// TwinCAT 3 PLC project Bohrmodell_SK1
// ProgramVersion: 3.1.4024.12
// libraries:
//   Tc2_EtherCAT, * (Beckhoff Automation GmbH)
//   Tc2_Standard, * (Beckhoff Automation GmbH)
//   Tc2_System, * (Beckhoff Automation GmbH)
//   Tc3_Module, * (Beckhoff Automation GmbH)
//   VisuSymbols,3.5.10.0,System
// project tree:
//   DUTs/ DUT_Motordaten.TcDUT, E_AmpelPhase.TcDUT, E_BMK.TcDUT, E_Step.TcDUT, ST_Test.TcDUT
//   / GlobalTextList.TcGTLO, PlcTask.TcTTO, TaktGen.TcTTO, Visualisierungsmanager.TcVMO (not stored)
//   GVLs/ GVL_Datenverarbeitung.TcGVL, GVL_GK_Automatikablauf.TcGVL, GVL_GlobalData.TcGVL, GVL_A1.TcGVL, GVL_C1.TcGVL, GVL_HMI.TcGVL
//   POUs/Ampelsteuerung/ DUT_AmpelConfig.TcDUT, E_Ampeln.TcDUT, FB_Ampel.TcPOU, GVL_Ampel.TcGVL, GVL_HMI_Ampel.TcGVL
//   POUs/Funktionen/ FB_Counter.TcPOU
//   POUs/HMI/ PRG_HMI.TcPOU
//   POUs/Mod01_Allgm/ FB_BA_Umschaltung_FUP.TcPOU, PRG_TaktGen.TcPOU, FB_BA_Umschaltung.TcPOU
//   POUs/Mod03_Diag/ FB_AdsLog.TcPOU
//   POUs/Mod20_Analog/ FB_Tank.TcPOU
//   POUs/ FB_StrukturieterText.TcPOU, POU_ST_FUP.TcPOU, PRG_MAIN.TcPOU
//   POUs/Geraete/ FB_Betriebsarten.TcPOU, FB_Motor.TcPOU
//   POUs/Mod10_FT/ FB_Antriebe.TcPOU, FB_Autoamtikablauf.TcPOU
//   POUs/Mod30/ FB_Refactoring.TcPOU, FB_RefDummy.TcPOU
//   POUs/TOOLS/ FB_Takt.TcPOU
//   VISUs/ Ampel.TcVIS, FP_Counter.TcVIS, Visualization.TcVIS
//   VISUs/Pages/ Page_2.TcVIS, Page_3.TcVIS
//   VISUs/Tempalte/ Visualization_1.TcVIS
// real-time tasks:
//   TASK PlcTask: cycle T#10ms, priority 6, ADS port 350
//   TASK TaktGen: cycle T#10ms, priority 8, ADS port 351
// I/O:
//   DEVICE Gerät 2 (EtherCAT), AmsNetId 172.16.0.8.3.1
//     Klemme 1 (EK1200) [EK1200-5000 EtherCAT Netzteil (2A E-Bus)]
//       -KF2 (EL1809) [EL1809 16K. Dig. Eingang 24V, 3ms]
//       Klemme 3 (EL1809) [EL1809 16K. Dig. Eingang 24V, 3ms]
//       Klemme 4 (EL2809) [EL2809 16K. Dig. Ausgang 24V, 0.5A]
//       Klemme 5 (EL2809) [EL2809 16K. Dig. Ausgang 24V, 0.5A]
//       Klemme 6 (EK1110) [EK1110 EtherCAT-Verlängerung]
//     Klemme 7 (EK1100) [EK1100 EtherCAT-Koppler (2A E-Bus)]
//       Klemme 8 (EL3062) [EL3062 2K.Ana. Eingang 0-10V]
//       Klemme 9 (EL4002) [EL4002 2K. Ana. Ausgang 0-10V, 12bit]
//       Klemme 10 (EL9011) [EL9011 Endklemme]
//     Box 20 (TB20 Coupler EtherCAT) [TB20 Coupler EtherCAT (600-185-1AA11)]
//       modules: Module 1 (8 DI - 600-210-0AH01), Module 2 (8 DO - 600-220-0AH01)
// variable links:
//   Bohrmodell_SK1/Bohrmodell_SK1 Instance <-> Device 2 (EtherCAT)/Term 1 (EK1200)/-KF2 (EL1809)
//     PlcTask Inputs/GVL_A1.GL1_B1_BG1 <-> Channel 9/GL1_B1_BG1
//     PlcTask Inputs/GVL_A1.GL2_B2_BG1 <-> Channel 10/GL2_B2_BG1
//     PlcTask Inputs/GVL_A1.GL3_B3_BG1 <-> Channel 11/Input
//     PlcTask Inputs/GVL_A1.TM1_B2_BG1 <-> Channel 12/Input
//     PlcTask Inputs/GVL_A1.TM1_B2_BG2 <-> Channel 13/Input
//     TaktGen Inputs/GVL_A1.GL1_B1_BQ1 <-> Channel 16/Input
//     TaktGen Inputs/GVL_A1.S01_C2_SF1 <-> Channel 14/Input
//     TaktGen Inputs/GVL_A1.S01_C3_SF1 <-> Channel 15/Input
//   Bohrmodell_SK1/Bohrmodell_SK1 Instance <-> Device 2 (EtherCAT)/Term 1 (EK1200)/Term 3 (EL1809)
//     PlcTask Inputs/GVL_C1.S01_C1_SF1 <-> Channel 1/S01_C1_SF1
//     PlcTask Inputs/GVL_C1.S01_C1_SF2 <-> Channel 2/S01_C1_SF2
//     PlcTask Inputs/GVL_C1.S01_C1_SF10 <-> Channel 10/Input
//     PlcTask Inputs/GVL_C1.S01_C1_SF11 <-> Channel 11/Input
//     PlcTask Inputs/GVL_C1.S01_C1_SF12 <-> Channel 12/Input
//     PlcTask Inputs/GVL_C1.S01_C1_SF13 <-> Channel 13/Input
//     PlcTask Inputs/GVL_C1.S01_C1_SF14 <-> Channel 14/Input
//     PlcTask Inputs/GVL_C1.S01_C1_SF16 <-> Channel 16/Input
//     PlcTask Inputs/GVL_C1.S01_C1_SF9 <-> Channel 9/Input
//     PlcTask Inputs/GVL_C1.S01_C1_SF3 <-> Channel 3/GVL_C1.S01_C1_SF3
//     TaktGen Inputs/GVL_C1.S01_C1_SF15 <-> Channel 15/Input
//     TaktGen Inputs/GVL_C1.S01_C1_SF6 <-> Channel 6/Input
//     TaktGen Inputs/GVL_C1.S01_C1_SF7 <-> Channel 7/Input
//     TaktGen Inputs/GVL_C1.S01_C1_SF8 <-> Channel 8/Input
//     TaktGen Inputs/GVL_C1.S01_C1_SF4 <-> Channel 4/GVL_C1.S01_C1_SF4
//     TaktGen Inputs/GVL_C1.S01_C1_SF5 <-> Channel 5/GVL_C1.S01_C1_SF5
//   Bohrmodell_SK1/Bohrmodell_SK1 Instance <-> Device 2 (EtherCAT)/Term 1 (EK1200)/Term 4 (EL2809)
//     PlcTask Outputs/GVL_A1.GL1_B1_MA1 <-> Channel 1/Output
//     PlcTask Outputs/GVL_A1.GL2_B2_MA1 <-> Channel 2/Output
//     PlcTask Outputs/GVL_A1.GL3_B3_MA1 <-> Channel 3/Output
//     PlcTask Outputs/GVL_A1.S01_C3_PF1 <-> Channel 11/Output
//     PlcTask Outputs/GVL_A1.S01_C3_PF2 <-> Channel 12/Output
//     PlcTask Outputs/GVL_A1.S01_C3_PF3 <-> Channel 13/Output
//     PlcTask Outputs/GVL_A1.S01_C3_PJ1 <-> Channel 15/Output
//     PlcTask Outputs/GVL_A1.TM1_B2_MA1 <-> Channel 4/Output
//     PlcTask Outputs/GVL_A1.TM1_B2_MA2_1 <-> Channel 5/Output
//     PlcTask Outputs/GVL_A1.TM1_B2_MA2_2 <-> Channel 6/Output
//     TaktGen Outputs/GVL_A1.S01_C2_PF1 <-> Channel 9/Output
//     TaktGen Outputs/GVL_A1.S01_C2_PF2 <-> Channel 10/Output
//     TaktGen Outputs/GVL_A1.S01_C3_PF4 <-> Channel 14/Output
//   Bohrmodell_SK1/Bohrmodell_SK1 Instance <-> Device 2 (EtherCAT)/Term 1 (EK1200)/Term 5 (EL2809)
//     PlcTask Outputs/GVL_C1.S01_C1_PF1 <-> Channel 1/Output
//     PlcTask Outputs/GVL_C1.S01_C1_PF10 <-> Channel 10/Output
//     PlcTask Outputs/GVL_C1.S01_C1_PF11 <-> Channel 11/Output
//     PlcTask Outputs/GVL_C1.S01_C1_PF15 <-> Channel 15/Output
//     PlcTask Outputs/GVL_C1.S01_C1_PF16 <-> Channel 16/Output
//     PlcTask Outputs/GVL_C1.S01_C1_PF2 <-> Channel 2/Output
//     PlcTask Outputs/GVL_C1.S01_C1_PF3 <-> Channel 3/Output
//     PlcTask Outputs/GVL_C1.S01_C1_PF4 <-> Channel 4/Output
//     PlcTask Outputs/GVL_C1.S01_C1_PF5 <-> Channel 5/Output
//     PlcTask Outputs/GVL_C1.S01_C1_PF6 <-> Channel 6/Output
//     PlcTask Outputs/GVL_C1.S01_C1_PF9 <-> Channel 9/Output
//     TaktGen Outputs/GVL_C1.S01_C1_PF12 <-> Channel 12/Output
//     TaktGen Outputs/GVL_C1.S01_C1_PF13 <-> Channel 13/Output
//     TaktGen Outputs/GVL_C1.S01_C1_PF14 <-> Channel 14/Output
//     TaktGen Outputs/GVL_C1.S01_C1_PF7 <-> Channel 7/Output
//     TaktGen Outputs/GVL_C1.S01_C1_PF8 <-> Channel 8/Output

CONFIGURATION Bohrmodell_SK1
    RESOURCE PLC ON TwinCAT3
        TASK PlcTask(INTERVAL := T#10ms, PRIORITY := 6);
        TASK TaktGen(INTERVAL := T#10ms, PRIORITY := 8);
        PROGRAM PRG_MAIN WITH PlcTask : PRG_MAIN;
        PROGRAM PRG_HMI WITH PlcTask : PRG_HMI;
        PROGRAM PRG_TaktGen WITH TaktGen : PRG_TaktGen;
    END_RESOURCE
END_CONFIGURATION

// ---- DUTs/DUT_Motordaten.TcDUT
TYPE DUT_Motordaten :
STRUCT
	Laufzeit : INT;
	Einschaltvorgange : UINT;
	Motorleistung : REAL;
	Motorstrom : REAL;
	Drehzahl : INT;
	ResetDisable : BOOL;
END_STRUCT
END_TYPE

// ---- DUTs/E_AmpelPhase.TcDUT
{attribute 'qualified_only'}
{attribute 'strict'}
TYPE E_AmpelPhase :
(
	INIT := 0,
	ROT,
	GRUEN,
	GELB,
	ROTGELB
);
END_TYPE

// ---- DUTs/E_BMK.TcDUT
{attribute 'qualified_only'}
{attribute 'strict'}
TYPE E_BMK :
(
	Band_1 := 1,
	Band_2 := 2,
	Band_3 := 3,
	Bohrer  := 4,	
	BW_FWD  := 5,
	BW_BWD  := 6
	
);
END_TYPE

// ---- DUTs/E_Step.TcDUT
{attribute 'qualified_only'}
{attribute 'strict'}
TYPE E_Step :
(
	START,
	STOP,
	DRILL_FWD,
	DRILL_BWD,
	FEED_IN,
	FEED_OUT,
	WAIT,
	IN_END_POS
	
);
END_TYPE

// ---- DUTs/ST_Test.TcDUT
TYPE ST_Test :
STRUCT
	var1: BOOL;
	var2: INT;
	VarArray: ARRAY [0..11] OF INT;
END_STRUCT
END_TYPE

// ---- POUs/Ampelsteuerung/DUT_AmpelConfig.TcDUT
TYPE DUT_AmpelConfig :
STRUCT
	tRot		:TIME; // Zet für die Rotphase
	tRotGelb	:TIME;	// Zeit für die RotGruenphase
	tGruen		:TIME;	// Zeit für die Gruenpahse
	tGelb		:TIME;	// Zeit für die Gelbphase
	active		: BOOL;
END_STRUCT
END_TYPE

// ---- POUs/Ampelsteuerung/E_Ampeln.TcDUT
{attribute 'qualified_only'}
{attribute 'strict'}
TYPE E_Ampeln :
(
	Lindesntrasse := 0,
	Hauptstrasse := 1,
	Nebenstrasse := 2
);
END_TYPE

// ---- GVLs/GVL_Datenverarbeitung.TcGVL
{attribute 'qualified_only'}
VAR_GLOBAL PERSISTENT
	a_Einschaltvorgaenge_Antrieb : ARRAY[1..6] OF UINT;
	a_Antriebe : ARRAY [1..6] OF DUT_Motordaten;
END_VAR

// ---- GVLs/GVL_GK_Automatikablauf.TcGVL
{attribute 'qualified_only'}
VAR_GLOBAL
b_A_Band_1 : BOOL;				// Signal für Band 1 im Automatikbetrieb
b_A_Band_2 : BOOL;				// Signal für Band 2 im Automatikbetrieb
b_A_Band_3 : BOOL;				// Signal für Band 3 im Automatikbetrieb
b_A_Bohrer : BOOL;				// Signal für den Bohrer im Automatikbetrieb
b_A_Bohrwerk_zurueck : BOOL;	// Signal für das Bohrwerk zurück im Automatikbetrieb
b_A_Bohrwerk_vor : BOOL;		// Signal für das Bohrwerk zurück im Automatikbetrieb
END_VAR

// ---- GVLs/GVL_GlobalData.TcGVL
{attribute 'qualified_only'}
VAR_GLOBAL
	
// Global
	b_BA_Hand		: BOOL;		// Betriebsart Hand
	b_BA_Auto		: BOOL;		// Betriebsart Automatik
	// Zahlenarray
	n_Array: ARRAY[0..1000] OF LINT;
	n_ArrayMax: ARRAY[0..65535] OF LINT;
	DataArray:	ARRAY[0..100] OF DINT;
	

END_VAR

// ---- GVLs/GVL_A1.TcGVL
{attribute 'qualified_only'}
VAR_GLOBAL

//
// Eingänge Bohrmodell
//=================================

GL1_B1_BG1		AT%I*	: BOOL;  // Belegtmeldung Station Zuführen [TRUE = belegt]
GL2_B2_BG1		AT%I*	: BOOL;  // Belegtmeldung Station Bearbeiten [TRUE = belegt]
GL3_B3_BG1		AT%I*	: BOOL;  //"Belegtmeldung Station Bereitstellen [TRUE = belegt]"
TM1_B2_BG1		AT%I*	: BOOL;  // "Endlage Bohrwerk hinten [TRUE = hinten]"
TM1_B2_BG2		AT%I*	: BOOL;  // "Endlage Bohrwerk vorne [TRUE = vorne]"
S01_C2_SF1		AT%I*	: BOOL;  // "Taster Station Zuführen "
S01_C3_SF1		AT%I*	: BOOL;  // "Taster Station Bereitstellen "
GL1_B1_BQ1		AT%I*	: BOOL;  // "Materialerkennung Station Zuführen [TRUE = Metall]"

//
// Ausgänge Bohrmodell
//=================================

GL1_B1_MA1		AT%Q*	: BOOL;  // "Motor Station Zuführen "
GL2_B2_MA1		AT%Q*	: BOOL;  // "Motor Station Bearbeiten"
GL3_B3_MA1		AT%Q*	: BOOL;  // "Motor Station Bereitstellen"
TM1_B2_MA1		AT%Q*	: BOOL;  // "Motor Bohrspindel"
TM1_B2_MA2_1	AT%Q*	: BOOL;	 // "Bohrschlitten zurück"
TM1_B2_MA2_2	AT%Q*	: BOOL;	 // "Bohrschlitten vor"        
S01_C2_PF1		AT%Q*	: BOOL;  // "Anzeige grün Station Zuführen "
S01_C2_PF2		AT%Q*	: BOOL;  // "Anzeige rot Station Zuführen "
S01_C3_PF1		AT%Q*	: BOOL;  // "Ampel rot Station Bereitstellen "
S01_C3_PF2		AT%Q*	: BOOL;  // "Ampel gelb Station Bereitstellen "
S01_C3_PF3		AT%Q*	: BOOL;  // "Ampel grün Station Bereitstellen "
S01_C3_PF4		AT%Q*	: BOOL;  // "Anzeige gelb Station Bereitstellen "
S01_C3_PJ1		AT%Q*	: BOOL;	 // "Signalgeber Hupe Station Bereitstellen "

END_VAR

// ---- GVLs/GVL_C1.TcGVL
{attribute 'qualified_only'}
VAR_GLOBAL

//
// Eingänge Bedienpult
//=================================

S01_C1_SF16		AT%I*   : BOOL; // Taster/Schalter Reset
S01_C1_SF15     AT%I*   : BOOL; // Taster/Schalter - Reserve
S01_C1_SF14     AT%I*   : BOOL; // Taster/Schalter BW vor EIN
S01_C1_SF13     AT%I*   : BOOL; // Taster/Schalter BW zurück EIN
S01_C1_SF12     AT%I*   : BOOL; // Taster/Schalter Bohrer EIN
S01_C1_SF11     AT%I*   : BOOL; // Taster/Schalter Band 3 EIN
S01_C1_SF10     AT%I*   : BOOL; // Taster/Schalter Band 2 EIN
S01_C1_SF9      AT%I*   : BOOL; // Taster/Schalter Band 1 EIN

S01_C1_SF8		AT%I*   : BOOL; // Taster/Schalter Quittieren
S01_C1_SF7      AT%I*   : BOOL; // Taster/Schalter 
S01_C1_SF6      AT%I*   : BOOL; // Taster/Schalter Rücksetzten
S01_C1_SF5      AT%I*   : BOOL; // Taster/Schalter Setzen
S01_C1_SF4      AT%I*   : BOOL; // Taster/Schalter Test IF
S01_C1_SF3      AT%I*   : BOOL; // Taster/Schalter Anwahl Automatik 
S01_C1_SF2      AT%I*   : BOOL; // Taster/Schalter Anwahl Hand
S01_C1_SF1      AT%I*   : BOOL; // Schalter Anlage EIN/AUS true=Anlage EIN

//
// Ausgänge Bedienpult
//=================================

S01_C1_PF16		AT%Q*	: BOOL; // Anzeige/LED  Warten Abnahme
S01_C1_PF15		AT%Q*	: BOOL; // Anzeige/LED  Stückzahl erreicht
S01_C1_PF14		AT%Q*	: BOOL; // Anzeige/LED  RS
S01_C1_PF13		AT%Q*	: BOOL; // Anzeige/LED  SR
S01_C1_PF12		AT%Q*	: BOOL; // Anzeige/LED  Test IF
S01_C1_PF11		AT%Q*	: BOOL; // Anzeige/LED  BA Auto EIN
S01_C1_PF10		AT%Q*	: BOOL; // Anzeige/LED  BA Hand EIN
S01_C1_PF9		AT%Q*	: BOOL; // Anzeige/LED  Anlage EIN

S01_C1_PF8		AT%Q*	: BOOL; // Anzeige/LED Störung
S01_C1_PF7		AT%Q*	: BOOL; // Anzeige/LED - Reserve
S01_C1_PF6		AT%Q*	: BOOL; // Anzeige/LED BW vor EIN
S01_C1_PF5		AT%Q*	: BOOL; // Anzeige/LED BW zurück EIN
S01_C1_PF4		AT%Q*	: BOOL; // Anzeige/LED Bohrer EIN
S01_C1_PF3		AT%Q*	: BOOL; // Anzeige/LED Band 3 EIN
S01_C1_PF2		AT%Q*	: BOOL; // Anzeige/LED Band 2 EIN
S01_C1_PF1		AT%Q*	: BOOL; // Anzeige/LED Band 1 EIN





END_VAR

// ---- GVLs/GVL_HMI.TcGVL
{attribute 'qualified_only'}
VAR_GLOBAL
	input_1 : BOOL;
	input_2	: BOOL;
	output_1:BOOL;
	
	//Countervariablen
	btn_CTU	: BOOL;
	btn_CTD	: BOOL;
	Counter	: DINT;
	
END_VAR

// ---- POUs/Ampelsteuerung/GVL_Ampel.TcGVL
{attribute 'qualified_only'}
VAR_GLOBAL
	config: ARRAY[0..20] OF DUT_AmpelConfig;
END_VAR

// ---- POUs/Ampelsteuerung/GVL_HMI_Ampel.TcGVL
{attribute 'qualified_only'}
VAR_GLOBAL
	
	LED_Rot	: BOOL;
	LED_Gelb: BOOL;
	LED_Gruen	: BOOL;
	
	btnReset	: BOOL;
	btnActive	: BOOL;
	
	bBlinktakt	: BOOL;
END_VAR

// ---- POUs/PRG_MAIN.TcPOU
PROGRAM PRG_MAIN
VAR
	
	fb_Antriebe : FB_Antriebe;
	fb_Betriebsart : FB_BA_Umschaltung;
	fbADSLogger		: FB_AdsLog;
	fbAmpel			: FB_Ampel;

END_VAR



fb_Betriebsart();
fb_Antriebe();
fbADSLogger();

fbAmpel(bBlinktakt := GVL_HMI_Ampel.bBlinktakt,
		btnReset:= GVL_HMI_Ampel.btnReset,
		btnActive := GVL_HMI_Ampel.btnActive,
		LED_ROT => GVL_HMI_Ampel.LED_Rot,
		LED_GELB => GVL_HMI_Ampel.LED_Gelb,
		LED_GRUEN => GVL_HMI_Ampel.LED_Gruen,
	config := GVL_Ampel.config[E_Ampeln.Lindesntrasse]);
		
GVL_A1.S01_C3_PF1 := fbAmpel.LED_ROT;
GVL_A1.S01_C3_PJ1 := fbAmpel.LED_ROT AND GVL_HMI_Ampel.bBlinktakt;
GVL_A1.S01_C3_PF2 := fbAmpel.LED_GELB;
GVL_A1.S01_C3_PF3 := fbAmpel.LED_GRUEN;

END_PROGRAM

// ---- POUs/Mod10_FT/FB_Antriebe.TcPOU
FUNCTION_BLOCK FB_Antriebe
VAR
	Antrieb_Band_1  : FB_Motor;
    Antrieb_Band_2	: FB_Motor;
    Antrieb_Band_3	: FB_Motor;
    Antrieb_Bohrer	: FB_Motor;
    Antrieb_BW_zurueck	: FB_Motor;
    Antrieb_BW_vor	:	FB_Motor;
	FB_Automatik_inst : FB_Autoamtikablauf;
END_VAR

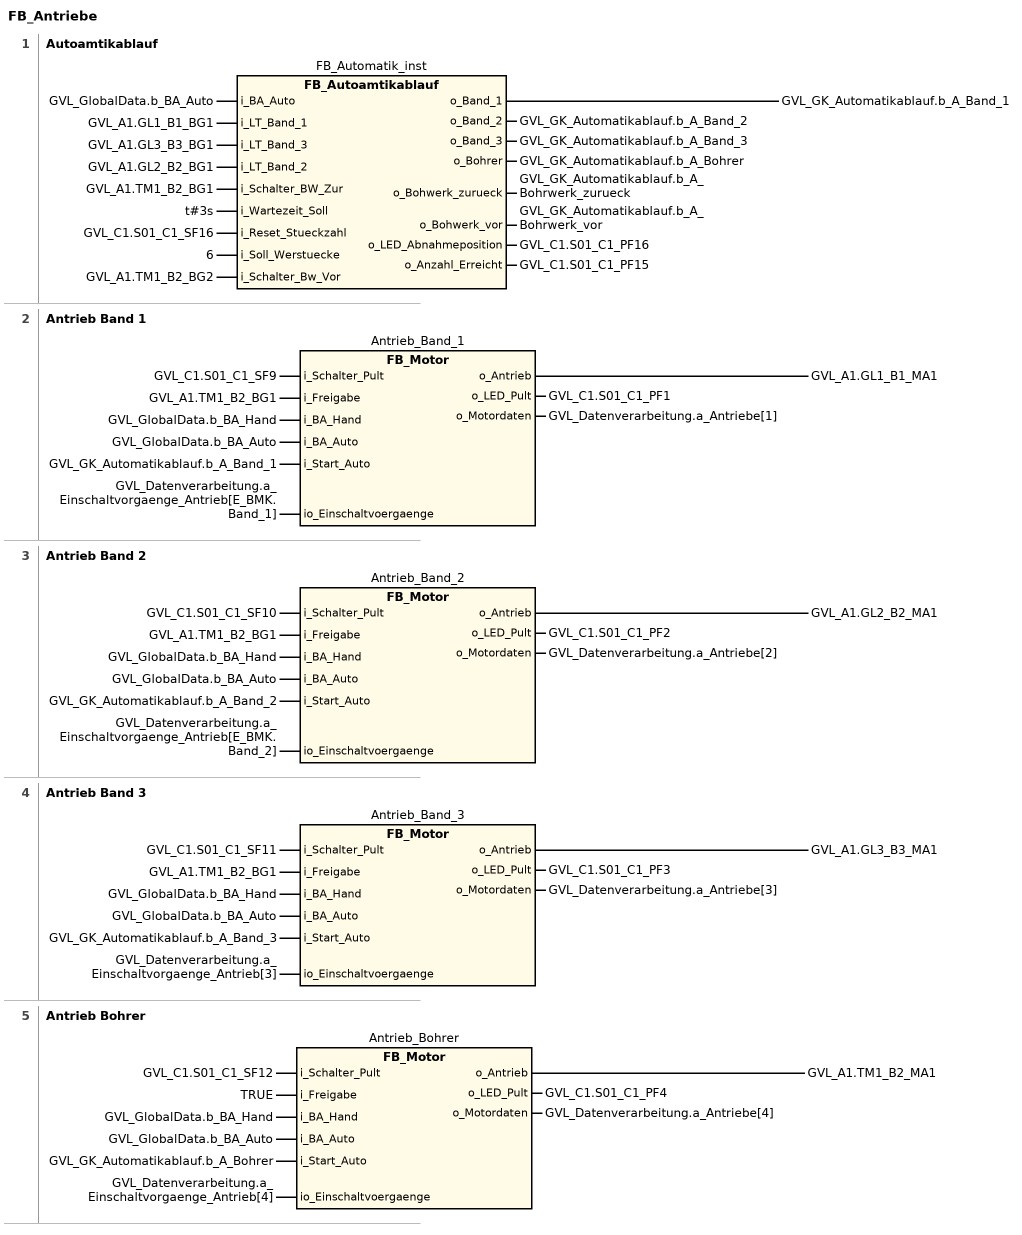
// NETWORK 1: Autoamtikablauf
FB_Automatik_inst(
    i_BA_Auto := GVL_GlobalData.b_BA_Auto,
    i_LT_Band_1 := GVL_A1.GL1_B1_BG1,
    i_LT_Band_3 := GVL_A1.GL3_B3_BG1,
    i_LT_Band_2 := GVL_A1.GL2_B2_BG1,
    i_Schalter_BW_Zur := GVL_A1.TM1_B2_BG1,
    i_Wartezeit_Soll := t#3s,
    i_Reset_Stueckzahl := GVL_C1.S01_C1_SF16,
    i_Soll_Werstuecke := 6,
    i_Schalter_Bw_Vor := GVL_A1.TM1_B2_BG2,
    o_Band_2 => GVL_GK_Automatikablauf.b_A_Band_2,
    o_Band_3 => GVL_GK_Automatikablauf.b_A_Band_3,
    o_Bohrer => GVL_GK_Automatikablauf.b_A_Bohrer,
    o_Bohwerk_zurueck => GVL_GK_Automatikablauf.b_A_Bohrwerk_zurueck,
    o_Bohwerk_vor => GVL_GK_Automatikablauf.b_A_Bohrwerk_vor,
    o_LED_Abnahmeposition => GVL_C1.S01_C1_PF16,
    o_Anzahl_Erreicht => GVL_C1.S01_C1_PF15); // FB_Autoamtikablauf
GVL_GK_Automatikablauf.b_A_Band_1 := FB_Automatik_inst.o_Band_1;

// NETWORK 2: Antrieb Band 1
Antrieb_Band_1(
    i_Schalter_Pult := GVL_C1.S01_C1_SF9,
    i_Freigabe := GVL_A1.TM1_B2_BG1,
    i_BA_Hand := GVL_GlobalData.b_BA_Hand,
    i_BA_Auto := GVL_GlobalData.b_BA_Auto,
    i_Start_Auto := GVL_GK_Automatikablauf.b_A_Band_1,
    io_Einschaltvoergaenge := GVL_Datenverarbeitung.a_Einschaltvorgaenge_Antrieb[E_BMK.Band_1],
    o_LED_Pult => GVL_C1.S01_C1_PF1,
    o_Motordaten => GVL_Datenverarbeitung.a_Antriebe[1]); // FB_Motor
GVL_A1.GL1_B1_MA1 := Antrieb_Band_1.o_Antrieb;

// NETWORK 3: Antrieb Band 2
Antrieb_Band_2(
    i_Schalter_Pult := GVL_C1.S01_C1_SF10,
    i_Freigabe := GVL_A1.TM1_B2_BG1,
    i_BA_Hand := GVL_GlobalData.b_BA_Hand,
    i_BA_Auto := GVL_GlobalData.b_BA_Auto,
    i_Start_Auto := GVL_GK_Automatikablauf.b_A_Band_2,
    io_Einschaltvoergaenge := GVL_Datenverarbeitung.a_Einschaltvorgaenge_Antrieb[E_BMK.Band_2],
    o_LED_Pult => GVL_C1.S01_C1_PF2,
    o_Motordaten => GVL_Datenverarbeitung.a_Antriebe[2]); // FB_Motor
GVL_A1.GL2_B2_MA1 := Antrieb_Band_2.o_Antrieb;

// NETWORK 4: Antrieb Band 3
Antrieb_Band_3(
    i_Schalter_Pult := GVL_C1.S01_C1_SF11,
    i_Freigabe := GVL_A1.TM1_B2_BG1,
    i_BA_Hand := GVL_GlobalData.b_BA_Hand,
    i_BA_Auto := GVL_GlobalData.b_BA_Auto,
    i_Start_Auto := GVL_GK_Automatikablauf.b_A_Band_3,
    io_Einschaltvoergaenge := GVL_Datenverarbeitung.a_Einschaltvorgaenge_Antrieb[3],
    o_LED_Pult => GVL_C1.S01_C1_PF3,
    o_Motordaten => GVL_Datenverarbeitung.a_Antriebe[3]); // FB_Motor
GVL_A1.GL3_B3_MA1 := Antrieb_Band_3.o_Antrieb;

// NETWORK 5: Antrieb Bohrer
Antrieb_Bohrer(
    i_Schalter_Pult := GVL_C1.S01_C1_SF12,
    i_Freigabe := TRUE,
    i_BA_Hand := GVL_GlobalData.b_BA_Hand,
    i_BA_Auto := GVL_GlobalData.b_BA_Auto,
    i_Start_Auto := GVL_GK_Automatikablauf.b_A_Bohrer,
    io_Einschaltvoergaenge := GVL_Datenverarbeitung.a_Einschaltvorgaenge_Antrieb[4],
    o_LED_Pult => GVL_C1.S01_C1_PF4,
    o_Motordaten => GVL_Datenverarbeitung.a_Antriebe[4]); // FB_Motor
GVL_A1.TM1_B2_MA1 := Antrieb_Bohrer.o_Antrieb;

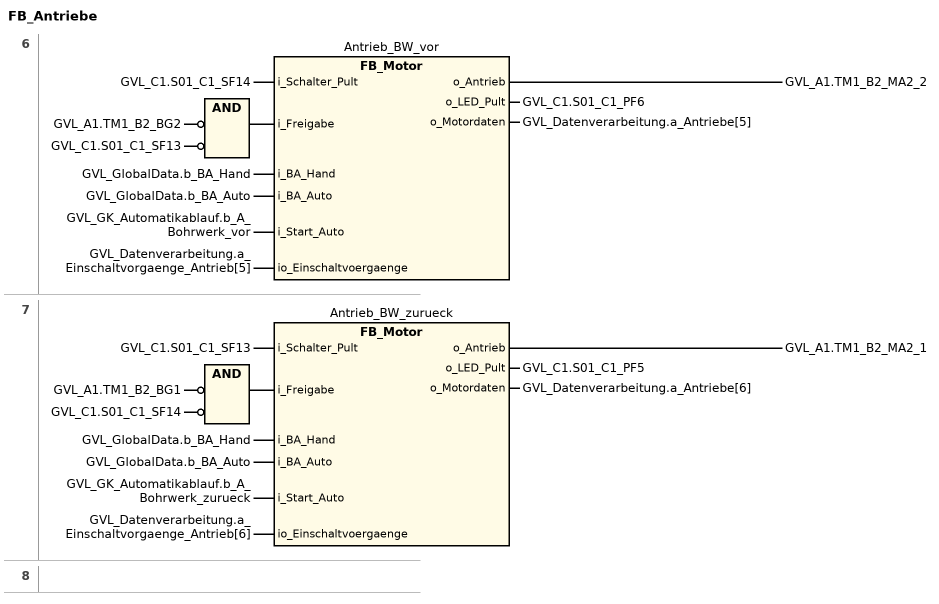
// NETWORK 6
Antrieb_BW_vor(
    i_Schalter_Pult := GVL_C1.S01_C1_SF14,
    i_Freigabe := NOT GVL_A1.TM1_B2_BG2 AND NOT GVL_C1.S01_C1_SF13,
    i_BA_Hand := GVL_GlobalData.b_BA_Hand,
    i_BA_Auto := GVL_GlobalData.b_BA_Auto,
    i_Start_Auto := GVL_GK_Automatikablauf.b_A_Bohrwerk_vor,
    io_Einschaltvoergaenge := GVL_Datenverarbeitung.a_Einschaltvorgaenge_Antrieb[5],
    o_LED_Pult => GVL_C1.S01_C1_PF6,
    o_Motordaten => GVL_Datenverarbeitung.a_Antriebe[5]); // FB_Motor
GVL_A1.TM1_B2_MA2_2 := Antrieb_BW_vor.o_Antrieb;

// NETWORK 7
Antrieb_BW_zurueck(
    i_Schalter_Pult := GVL_C1.S01_C1_SF13,
    i_Freigabe := NOT GVL_A1.TM1_B2_BG1 AND NOT GVL_C1.S01_C1_SF14,
    i_BA_Hand := GVL_GlobalData.b_BA_Hand,
    i_BA_Auto := GVL_GlobalData.b_BA_Auto,
    i_Start_Auto := GVL_GK_Automatikablauf.b_A_Bohrwerk_zurueck,
    io_Einschaltvoergaenge := GVL_Datenverarbeitung.a_Einschaltvorgaenge_Antrieb[6],
    o_LED_Pult => GVL_C1.S01_C1_PF5,
    o_Motordaten => GVL_Datenverarbeitung.a_Antriebe[6]); // FB_Motor
GVL_A1.TM1_B2_MA2_1 := Antrieb_BW_zurueck.o_Antrieb;

// NETWORK 8

END_FUNCTION_BLOCK

// ---- POUs/Geraete/FB_Motor.TcPOU
FUNCTION_BLOCK FB_Motor
VAR_INPUT
	i_Schalter_Pult: BOOL; 	// Schalter für die Manuelle bedienung des Motors über das Pult
	i_Freigabe : BOOL;		// Freigabe für das Ansteuern des Motors (TRUE für Freigabe FALSE für Verriegelung)
	i_BA_Hand: BOOL;		// Betriebsart Hand aktiv
	
	// Betriebsart Autoamtik aktiv
	i_BA_Auto: BOOL;
	// Start des Antriebs in Automatikbetrieb
	i_Start_Auto: BOOL;
END_VAR
VAR_OUTPUT
	o_Antrieb : BOOL; 		// Ausgang für die Antriebsansteuerung (TRUE = Motor EIN)
	o_LED_Pult : BOOL;		// Anzeige für Motor EIN
	o_Motordaten: DUT_Motordaten;
END_VAR

VAR
	FM_Einschaltvorgaenge : R_TRIG;  // Postive Flankenabfrage
END_VAR

VAR_TEMP
	t_Antrieb : BOOL;		// Variable als Zwischenspeicher des Antriebssignals
	re_MotorEin : BOOL;
END_VAR

VAR_IN_OUT
	io_Einschaltvoergaenge: UINT;
END_VAR

// Bildung des Steuersignals für Motoransteuerung
t_Antrieb := ((i_BA_Hand AND i_Schalter_Pult)
				OR (i_BA_Auto AND i_Start_Auto)) AND i_Freigabe;	
o_Antrieb := t_Antrieb;							// Zuweisung des Steuersignals an den Ausgang Antrieb
o_LED_Pult := t_Antrieb;						// Zweisung des Steuersignals an die Meldeleuchte

FM_Einschaltvorgaenge(CLK:=t_Antrieb , Q=> );

IF FM_Einschaltvorgaenge.Q THEN
	io_Einschaltvoergaenge := io_Einschaltvoergaenge +1;
END_IF


o_Motordaten.Einschaltvorgange := io_Einschaltvoergaenge;

END_FUNCTION_BLOCK

// ---- POUs/Mod10_FT/FB_Autoamtikablauf.TcPOU
FUNCTION_BLOCK FB_Autoamtikablauf
VAR_INPUT
	i_BA_Auto : BOOL;
	i_LT_Band_1 : BOOL;
	i_LT_Band_3 : BOOL;
	i_LT_Band_2 : BOOL;
	i_Schalter_BW_Zur : BOOL;
	i_Schalter_Bw_Vor : BOOL;
	i_Wartezeit_Soll: TIME;
	
	i_Reset_Stueckzahl: BOOL;
	i_Soll_Werstuecke: USINT;
END_VAR
VAR_OUTPUT
		
	o_Band_1 : BOOL;
	o_Band_2 : BOOL;
	o_Band_3 : BOOL;
	o_Bohrer : BOOL;
	o_Bohwerk_zurueck : BOOL;
	o_Bohwerk_vor : BOOL;
	o_LED_Abnahmeposition : BOOL;
	
	o_Anzahl_Erreicht: BOOL;
END_VAR
VAR
	SchrittNr : INT := 0;		// INndexvariable / Schrittnummer
	TON_Einlaufverzoegerung : TON;
	//eStp : (INIT, INFEED, BW_Fwd,BW_Bwd,OUTFEED,IN_ENDPOS,WAIT  );
	CTU_Werkstueckzaehler : CTU;
	eStep : (INIT, FEED_IN, DRILL_FWD, DRILL_BWD,FEED_OUT,IN_END_POS, WAIT, ERROR);
	
END_VAR

VAR_TEMP
	t_Wartezeit_abgelaufen : BOOL;
END_VAR

// Rücksetzen des Schrittnummer wenn Automatik nicht aktiv.

IF NOT i_BA_Auto THEN
		o_Band_1 := 0;
		o_Band_2 := 0;
		o_Band_3 := 0;
		o_Bohrer := 0;
		o_Bohwerk_vor := 0;
		o_Bohwerk_zurueck := 0;
		o_LED_Abnahmeposition := 0;
		SchrittNr := 0;
END_IF

// Hier ein Bereich für den Code
/////////////////////

		CASE SchrittNr OF
			
			INIT:
			IF i_BA_Auto AND NOT i_Schalter_BW_Zur THEN
				o_Bohwerk_zurueck := 1;
			ELSIF i_BA_Auto AND i_Schalter_BW_Zur THEN
				o_Bohwerk_zurueck := 0;
				SchrittNr := FEED_IN ;
			ELSE;
			END_IF
			
			FEED_IN:  // Transport von Pos 1 nach Pos 2
			TON_Einlaufverzoegerung(IN:=i_BA_Auto AND i_LT_Band_1 AND NOT CTU_Werkstueckzaehler.Q ,
									 PT:= i_Wartezeit_Soll,
									 Q=> t_Wartezeit_abgelaufen,
									 ET=> );
									 
		
									 
			//IF  t_Wartezeit_abgelaufen THEN
			IF  t_Wartezeit_abgelaufen THEN
				o_Band_1 := 1;
				o_Band_2 := 1;
				o_Band_3 := 0;
				o_Bohrer := 0;
				o_Bohwerk_vor := 0;
				o_Bohwerk_zurueck := 0;
				SchrittNr := DRILL_FWD ;
			ELSE;
			END_IF
			
			DRILL_FWD: // Bohrwerk vor Fahren
			IF i_BA_Auto AND i_LT_Band_2 THEN
				o_Band_1 := 0;
				o_Band_2 := 0;
				o_Band_3 := 0;
				o_Bohrer := 1;
				o_Bohwerk_vor := 1;
				o_Bohwerk_zurueck := 0;
				SchrittNr := DRILL_BWD ;
			ELSE;
			END_IF
			
			
			DRILL_BWD: // Bohrwerk zurück Fahren
			IF i_BA_Auto AND i_Schalter_Bw_Vor THEN
				o_Band_1 := 0;
				o_Band_2 := 0;
				o_Band_3 := 0;
				o_Bohrer := 1;
				o_Bohwerk_vor := 0;
				o_Bohwerk_zurueck := 1;
				SchrittNr := FEED_OUT ;
			ELSE;
			END_IF
			
			FEED_OUT: // Transport von Pos 2 nach Pos 3
			IF i_BA_Auto AND i_Schalter_BW_Zur THEN
				o_Band_1 := 0;
				o_Band_2 := 1;
				o_Band_3 := 1;
				o_Bohrer := 0;
				o_Bohwerk_vor := 0;
				o_Bohwerk_zurueck := 0;
				SchrittNr := IN_END_POS ;
			ELSE;
			END_IF
			
			IN_END_POS: // Abnahmepostion erreicht
			IF i_BA_Auto AND i_LT_Band_3 THEN
				o_Band_1 := 0;
				o_Band_2 := 0;
				o_Band_3 := 0;
				o_Bohrer := 0;
				o_Bohwerk_vor := 0;
				o_Bohwerk_zurueck := 0;
				o_LED_Abnahmeposition := 1;
				SchrittNr := WAIT ;
			ELSE;
			END_IF
			
			WAIT: // Wartena auf Abnahme
			IF i_BA_Auto AND NOT i_LT_Band_3 THEN
				o_LED_Abnahmeposition := 0;
				SchrittNr := INIT ;
			ELSE;
			END_IF
		
		ELSE  // Sicherheitsabfrage falls Zähler nicht plausibel
				o_Band_1 := 0;
				o_Band_2 := 0;
				o_Band_3 := 0;
				o_Bohrer := 0;
				o_Bohwerk_vor := 0;
				o_Bohwerk_zurueck := 0;
				
		END_CASE

CTU_Werkstueckzaehler(
	CU:= i_BA_Auto AND i_LT_Band_3 , 
	RESET:= i_Reset_Stueckzahl, 
	PV:= i_Soll_Werstuecke, 
	Q=> o_Anzahl_Erreicht, 
	CV=> );

END_FUNCTION_BLOCK

// ---- POUs/Mod01_Allgm/FB_BA_Umschaltung.TcPOU
FUNCTION_BLOCK FB_BA_Umschaltung
VAR_INPUT
END_VAR
VAR_OUTPUT
END_VAR
VAR
	FB_BA_Hand : FB_Betriebsarten;
	FB_BA_Auto : FB_Betriebsarten;
END_VAR

// Betriebsartenumdschaltung
//==========================
// 15.02.2023 J.Friesen
// Wenn der Hauptschalter "Anlage Ein" Betätigt ist soll es möglich sein die Betriebsarten
// zu aktiveiren. Die Betriebsarten sollen gegen einander verriegelt sein so, dass
// das Aktiveren beider Betriebsarten gleichzeitig nicht möglich sein soll. 


// Aufruf der Betriebsartenumschaltung für Automatikbetrieb
FB_BA_Auto(i_S_Analge_ein:= GVL_C1.S01_C1_SF1,	
			i_T_BA_ein:=  GVL_C1.S01_C1_SF3 ,
			i_T_BA_aus:=  GVL_C1.S01_C1_SF2,	
			o_BA=> GVL_GlobalData.b_BA_Auto);
			

// Aufruf der Betriesartenumschaltung für handbetrieb			
FB_BA_Hand(	i_S_Analge_ein:= GVL_C1.S01_C1_SF1 ,
 			i_T_BA_ein:=  GVL_C1.S01_C1_SF2,
			i_T_BA_aus:=  GVL_C1.S01_C1_SF3,
			o_BA=> GVL_GlobalData.b_BA_Hand);
			
			
// Signalzuweisung zu Pult Meldeleuchten
//=========================================		
	GVL_C1.S01_C1_PF9 := GVL_C1.S01_C1_SF1;  		// Zuweisung Meldeleuchte PULT
	GVL_C1.S01_C1_PF10 := GVL_GLobalData.b_BA_Hand;	// Zuweisung Meldleuchte Pult BA Hand
	GVL_C1.S01_C1_PF11 := GVL_GLobalData.b_BA_Auto;	// Zuweisung Meldeleuchte Pult BA Automatik

END_FUNCTION_BLOCK

// ---- POUs/Geraete/FB_Betriebsarten.TcPOU
FUNCTION_BLOCK FB_Betriebsarten

VAR_INPUT
	i_S_Analge_ein	: BOOL;  // Signal, dass die Anlage aktiv ist
	i_T_BA_ein		: BOOL;		// Signal für das aktivieren der Betriebsart
	i_T_BA_aus		: BOOL;		// Signal für das deaktivieren der Betriebsart
END_VAR
VAR_OUTPUT
	o_BA			: BOOL;  // Ausgang für die aktive Betriebsart
END_VAR
VAR
END_VAR

IF NOT i_S_Analge_ein OR i_T_BA_aus THEN		// Abfrage Anlae ein und Verriegelung
	o_BA := FALSE;								// Betriebsart ausschalten
ELSIF i_T_BA_ein THEN							// Abfrage Taster Betriebsart
	o_BA := TRUE;								// Betreibsart einschalten
END_IF

END_FUNCTION_BLOCK

// ---- POUs/Mod03_Diag/FB_AdsLog.TcPOU
FUNCTION_BLOCK FB_AdsLog
VAR_INPUT
END_VAR
VAR_OUTPUT
END_VAR
VAR
	reBtnReset	: R_TRIG;						// Flankenerkennng für Meldeauslösung
	udiAdsLogResStr	: DINT;						// Aufrufergebnis 0 = i.O. oder Fehlercode
	strMessageVariable	: STRING := 'Reset';	// Variabler Meldetext
	
END_VAR


reBtnReset(CLK:=GVL_C1.S01_C1_SF16);
IF reBtnReset.Q THEN
	udiAdsLogResStr:= ADSLOGSTR(msgCtrlMask:=	ADSLOG_MSGTYPE_WARN 
												OR ADSLOG_MSGTYPE_LOG 
												OR ADSLOG_MSGTYPE_MSGBOX ,
												 msgFmtStr:= 'Betätigte Taste: %s',
												strArg:=strMessageVariable );
END_IF;

END_FUNCTION_BLOCK

// ---- POUs/Ampelsteuerung/FB_Ampel.TcPOU
FUNCTION_BLOCK FB_Ampel
VAR_INPUT
	btnReset	: BOOL;
	btnActive	: BOOL;
	bBlinktakt	: BOOL;
	config	: DUT_AmpelConfig;
END_VAR
VAR_OUTPUT
	LED_ROT	: BOOL;
	LED_GELB:	BOOL;
	LED_GRUEN: 	BOOL;
END_VAR
VAR
	state	: E_AmpelPhase := E_AmpelPhase.INIT;
	tRot	: TON;  // Leuchtdauer Rot
	tRotGelb	: TON; // Leuchtdauer RotGelb
	tGruen	: TON;		// Leuchtaduer Gruen
	tGelb	: TON;		// Leuchtdauer Gelb
END_VAR


CASE state OF
	E_AmpelPhase.INIT:
			LED_ROT	:= FALSE;
			LED_GELB := bBlinktakt;
			LED_GRUEN := FALSE;
	
	E_AmpelPhase.ROT:
			LED_ROT	:= TRUE;
			LED_GELB := FALSE;
			LED_GRUEN := FALSE;
			IF tRot.Q THEN
				state := E_AmpelPhase.ROTGELB;
			END_IF
			
	E_AmpelPhase.ROTGELB:
			LED_ROT	:= TRUE;
			LED_GELB := TRUE;
			LED_GRUEN := FALSE;
			IF tRotGelb.Q THEN
				state := E_AmpelPhase.GRUEN;
			END_IF
			
	E_AmpelPhase.GRUEN:
			LED_ROT	:= FALSE;
			LED_GELB := FALSE;
			LED_GRUEN := TRUE;
			IF tGruen.Q THEN
				state := E_AmpelPhase.GELB;
			END_IF
			
	E_AmpelPhase.GELB:
			LED_ROT	:= FALSE;
			LED_GELB := TRUE;
			LED_GRUEN := FALSE;
			IF tGelb.Q THEN
				state := E_AmpelPhase.ROT;
			END_IF
ELSE
			LED_Gelb := bBlinktakt;
			LED_ROT	:= FALSE;
			LED_GRUEN := FALSE;
END_CASE

IF btnReset THEN
	state := E_AmpelPhase.INIT;
	ELSE ;
END_IF

IF btnActive AND (state = E_AmpelPhase.INIT) THEN
	state := E_AmpelPhase.ROT;
END_IF


// Timer

tRot(	IN:=(state = E_AmpelPhase.ROT),
		PT := config.tRot);
		
tRotGelb(	IN:=(state = E_AmpelPhase.ROTGELB),
		PT := config.tRotGelb);
		
tGruen(	IN:=(state = E_AmpelPhase.GRUEN),
		PT := config.tGruen);

tGelb(	IN:=(state = E_AmpelPhase.GELB),
		PT := config.tGelb);

END_FUNCTION_BLOCK

// ---- POUs/HMI/PRG_HMI.TcPOU
PROGRAM PRG_HMI
VAR
	counter	: FB_Counter;
END_VAR

GVL_HMI.output_1:=  GVL_HMI.input_1 AND GVL_HMI.input_2;

counter(CTU:=GVL_HMI.btn_CTU ,
		CTD:=GVL_HMI.btn_CTD , 
		Step:= 1, 
		Value:= GVL_HMI.Counter);

END_PROGRAM

// ---- POUs/Funktionen/FB_Counter.TcPOU
FUNCTION_BLOCK FB_Counter
VAR_INPUT
	CTU	:BOOL;		// Eingang zum hoch zählen
	CTD	:BOOL;		// Eingang zum abwärts zählen
	Step:INT := 1;		// Schrittweite
END_VAR
VAR_IN_OUT
	Value: DINT;	// Zählwert
END_VAR
VAR // added by the converter: edge detectors and wires of the graphical bodies
    _rt1, _rt2 : R_TRIG;
END_VAR

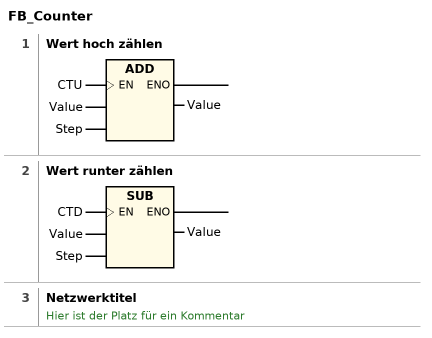
// NETWORK 1: Wert hoch zählen
_rt1(CLK := CTU);
IF _rt1.Q THEN Value := Value + Step; END_IF

// NETWORK 2: Wert runter zählen
_rt2(CLK := CTD);
IF _rt2.Q THEN Value := Value - Step; END_IF

// NETWORK 3: Netzwerktitel
// Hier ist der Platz für ein Kommentar

END_FUNCTION_BLOCK

// ---- POUs/Mod01_Allgm/PRG_TaktGen.TcPOU
PROGRAM PRG_TaktGen
VAR
	fb_TaktGen	: FB_Takt;
END_VAR

fb_TaktGen();

END_PROGRAM

// ---- POUs/TOOLS/FB_Takt.TcPOU
FUNCTION_BLOCK FB_Takt
VAR_INPUT
END_VAR
VAR_OUTPUT
END_VAR
VAR
	Timer_1s : TON; // timer für den Takt
	Timer_500ms	:TON;	//Timer für Ampelblinktakt
	Takt_1s	: BOOL;	// Tooglevariable
	
END_VAR

Timer_1s(IN:=NOT Timer_1s.Q ,
		 PT:=T#1S );
		 
Takt_1s := Takt_1s XOR Timer_1s.Q;

//Timer für Ampelblinktakt
Timer_500ms(IN:=NOT Timer_500ms.Q ,
		 	PT:=T#600MS );
			
GVL_HMI_Ampel.bBlinktakt := GVL_HMI_Ampel.bBlinktakt 
							XOR Timer_500ms.Q;

END_FUNCTION_BLOCK

// ---- POUs/Mod01_Allgm/FB_BA_Umschaltung_FUP.TcPOU
FUNCTION_BLOCK FB_BA_Umschaltung_FUP
VAR_INPUT
END_VAR
VAR_OUTPUT
END_VAR
VAR
	FB_BA_Hand : FB_Betriebsarten;
	FB_BA_Auto : FB_Betriebsarten;
END_VAR

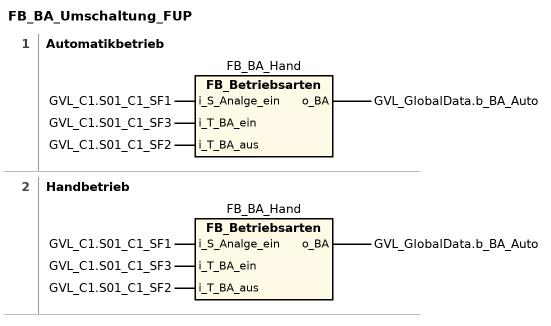
// NETWORK 1: Automatikbetrieb
FB_BA_Hand(
    i_S_Analge_ein := GVL_C1.S01_C1_SF1,
    i_T_BA_ein := GVL_C1.S01_C1_SF3,
    i_T_BA_aus := GVL_C1.S01_C1_SF2); // FB_Betriebsarten
GVL_GlobalData.b_BA_Auto := FB_BA_Hand.o_BA;

// NETWORK 2: Handbetrieb
FB_BA_Hand(
    i_S_Analge_ein := GVL_C1.S01_C1_SF1,
    i_T_BA_ein := GVL_C1.S01_C1_SF3,
    i_T_BA_aus := GVL_C1.S01_C1_SF2); // FB_Betriebsarten
GVL_GlobalData.b_BA_Auto := FB_BA_Hand.o_BA;

END_FUNCTION_BLOCK

// ---- POUs/Mod20_Analog/FB_Tank.TcPOU
FUNCTION_BLOCK FB_Tank
VAR_INPUT
	i_Fuellstand : INT;
END_VAR
VAR_OUTPUT
	o_Fuellstand : INT;
	o_Drehzahl 	: INT;
END_VAR
VAR
	g_Fuellstand : REAL; // Normierter Füllstandswert
	g_Drehzahl : REAL;  	// Normierter Drehzahlwert
	
END_VAR


g_Fuellstand := scale_in(
	input:= i_Fuellstand, 
	DV_min:= 0, 
	DV_max:= 32767, 
	LOW_Lim:= 0, 
	High_Lim:= 125);
	
o_Fuellstand := scale_out(
	input:= g_Fuellstand, 
	DV_min:= 0, 
	DV_max:= 32767, 
	LOW_Lim:= 0, 
	High_Lim:= 125);
	
	
	
o_Drehzahl := scale_out(
	input:= g_Drehzahl, 
	DV_min:= 0, 
	DV_max:= 32767, 
	LOW_Lim:= 0, 
	High_Lim:= 100);
	
	
	
	
	
	
	
	
	
	
	
	
	
	
	
	
	
	
	
	
// Motorsteuerung
IF g_Fuellstand >= 50 AND g_Fuellstand < 100 THEN
	g_Drehzahl := 50;
ELSIF g_Fuellstand >= 100 THEN
	g_Drehzahl := 100;
ELSE
	g_Drehzahl := 0;
END_IF

END_FUNCTION_BLOCK

// ---- POUs/FB_StrukturieterText.TcPOU
FUNCTION_BLOCK FB_StrukturieterText
VAR_INPUT
END_VAR
VAR_OUTPUT
END_VAR
VAR
	nCounter: INT := 0;
	nCounterSav: INT := 0;
	reCount	: R_TRIG;
	ForceCheck	: BOOL;
	Ergebnis : INT ;
	Wert1	: INT;
	Wert2	: INT;
	Motor1	:BOOL;
	Motor2	:BOOL;
	Zylinder:BOOL;
	Zylinder2:BOOL;
	step:int;
	
	Bedingung: BOOL;
	Anweisungen	:BOOL;
	Anweisungen2: BOOL;
	Anweisungen3: BOOL;
END_VAR







Ergebnis := Wert1 + Wert2;


IF Bedingung THEN
	Anweisungen;
ELSIF
	Anweisungen2;
ELSE
	Anweisungen3;
END_IF





IF Bedingung THEN
	Anweisungen;
ELSIF
	Anweisungsblock2;
ELSE
	Anweisung
END_IF













CASE step OF	
	1:	Motor1:= TRUE;
		Motor2:= FALSE;
		
	2,7:	Motor1:= FALSE;
			Motor2:= TRUE;
		
	8..12:	Motor1:= TRUE;
			Motor2:= TRUE;
ELSE
		Motor1:= FALSE;
		Motor2:= FALSE;
END_CASE












nCounter := 5000;
nCounter := nCounter + 1;
nCounter := nCounter + 1;
nCounter := nCounter + 1;
nCounter := nCounter + 1;
nCounter := nCounter + 1;
nCounter := nCounter + 1;
nCounter := nCounter + 1;

//IF nCounter = 600 THEN 
//	ForceCheck := TRUE;
//ELSE
//	ForceCheck := FALSE;
//END_IF

reCount(CLK:=PRG_TaktGen.fb_Taktmerker.Takt_1s);
IF reCount.Q THEN
	nCounter := nCounter + 1;
	nCounter := nCounter + 1;
	nCounter := nCounter + 1;
	nCounter := nCounter + 1;
	nCounter := nCounter + 1;
	nCounter := nCounter + 1;
	nCounter := nCounter + 1;
	nCounterSav := nCounter;
	
END_IF

nCounter := nCounter;
IF NOT PRG_TaktGen.fb_Taktmerker.Takt_1s THEN
	nCounterSav := 0;
END_IF

END_FUNCTION_BLOCK

// ---- POUs/Mod30/FB_Refactoring.TcPOU
FUNCTION_BLOCK FB_Refactoring
VAR_INPUT
	i_a  :BOOL;
    i_b  :BOOL;
    i_c  :BOOL;
    i_d  :BOOL;
    i_e  :BOOL;
    i_f  :BOOL;
   
END_VAR
VAR_OUTPUT
	q_a   :BOOL;
    q_b   :BOOL;
    q_c   :BOOL;
END_VAR
VAR
	ref_Dummy	: FB_RefDummy;
END_VAR

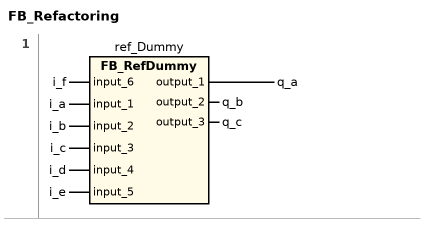
// NETWORK 1
ref_Dummy(
    input_6 := i_f,
    input_1 := i_a,
    input_2 := i_b,
    input_3 := i_c,
    input_4 := i_d,
    input_5 := i_e,
    output_2 => q_b,
    output_3 => q_c); // FB_RefDummy
q_a := ref_Dummy.output_1;

END_FUNCTION_BLOCK

// ---- POUs/Mod30/FB_RefDummy.TcPOU
FUNCTION_BLOCK FB_RefDummy
VAR_INPUT
	input_6  :BOOL;

	input_1  :BOOL;
    input_2  :BOOL;
    input_3  :BOOL;
    input_4  :BOOL;
    input_5  :BOOL;
    
END_VAR
VAR_OUTPUT

	output_1  :BOOL;
    output_2  :BOOL;
    output_3  :BOOL;

END_VAR
VAR
END_VAR

// NETWORK 1

END_FUNCTION_BLOCK

// ---- POUs/POU_ST_FUP.TcPOU
FUNCTION_BLOCK POU_ST_FUP
VAR_INPUT
END_VAR
VAR_OUTPUT
END_VAR
VAR
END_VAR

// NETWORK 1

END_FUNCTION_BLOCK

// ---- GlobalTextList.TcGTLO
TEXTLIST GlobalTextList
  442 = '%d'
  183 = '%s'
  58 = 'Active'
  191 = 'asdf'
  984 = 'CTD'
  592 = 'CTU'
  10 = 'Der Zähler wird um eins Inkrementiert'
  582 = 'Freigabe'
  676 = 'mm'
  194 = 'Reset'
  605 = 'Signalbez'
  737 = 'Text'
  689 = 'Werkstücke'
  739 = 'Zählwert %d'
END_TEXTLIST

// ---- VISUs/Ampel.TcVIS
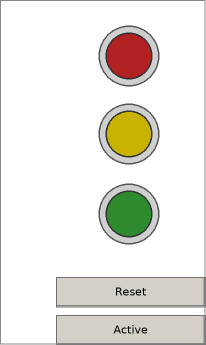
VISUALIZATION Ampel  // 206x345
    Lamp1 (94,21 70x70), variable: GVL_HMI_Ampel.LED_Rot, style: Lamp-Lamp1-Red
    Lamp1 (94,99 70x70), variable: GVL_HMI_Ampel.LED_Gelb, style: Lamp-Lamp1-Yellow
    Lamp1 (94,179 70x70), variable: GVL_HMI_Ampel.LED_Gruen, style: Lamp-Lamp1-Green
    Button (56,277 150x30), "Reset"
        tap GVL_HMI_Ampel.btnReset
    Button (56,315 150x30), "Active"
        tap GVL_HMI_Ampel.btnActive
END_VISUALIZATION

// ---- VISUs/FP_Counter.TcVIS
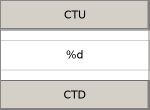
VISUALIZATION FP_Counter  // 150x110
VAR_IN_OUT
	o_CTU		: BOOL;
	o_CTD		: BOOL;
END_VAR

VAR_INPUT
	ctnValue	: INT;
END_VAR
    Group (0,0 150x110)
        Button (0,0 150x30), "CTU"
            tap btnCTU
        Button (0,80 150x30), "CTD"
            tap btuCTD
        Textfield (0,40 150x30), "%d", text variable: ctnValue
END_VISUALIZATION

// ---- VISUs/Pages/Page_2.TcVIS
VISUALIZATION Page_2  // 2x2
END_VISUALIZATION

// ---- VISUs/Pages/Page_3.TcVIS
VISUALIZATION Page_3  // 2x2
END_VISUALIZATION

// ---- VISUs/Tempalte/Visualization_1.TcVIS
VISUALIZATION Visualization_1  // 2x2
END_VISUALIZATION

// ---- VISUs/Visualization.TcVIS
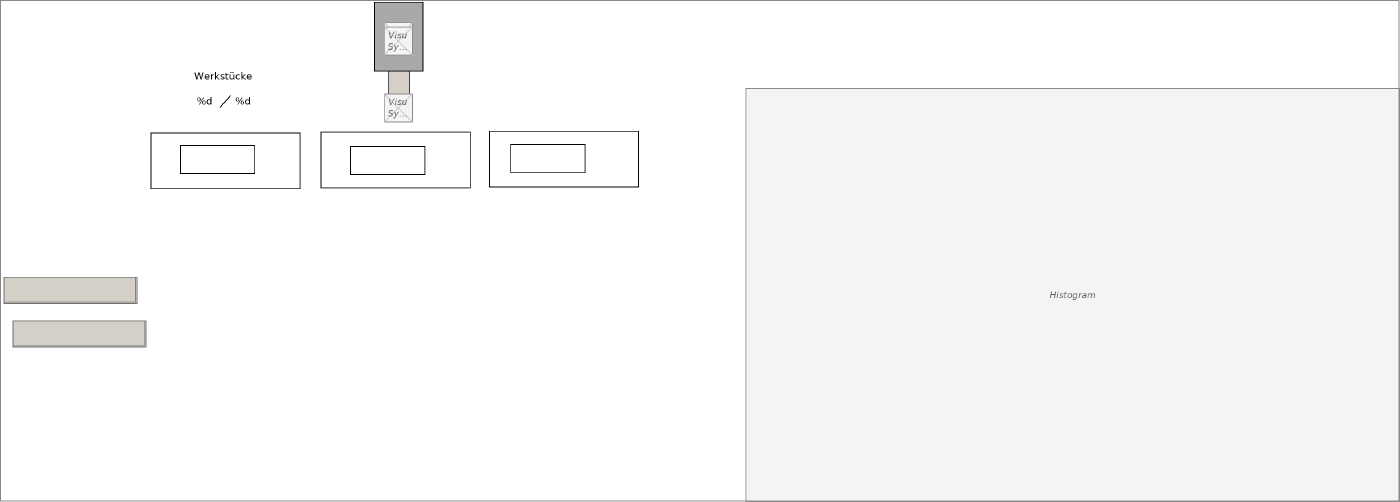
VISUALIZATION Visualization  // 1572x564
    RoundedRectangle (169,149 168x63), colour toggle: GVL_HMI.Status_Band_3, colour variable: 16#ff999999
        p3450524324: 16#00555555
        p2167032090: 16#ff00FF00
        p3092690914: 16#00555555
    RoundedRectangle (360,148 168x63), colour toggle: GVL_HMI.Status_Band_2, colour variable: 16#ff999999
        p3450524324: 16#00555555
        p2167032090: 16#ff00FF00
        p3092690914: 16#00555555
    RoundedRectangle (549,147 168x63), colour toggle: GVL_IO.A_Band_1, colour variable: 16#ff999999
        p2167032090: 16#ff00FF00
        p3450524324: 16#00555555
        p3092690914: 16#00555555
    RoundedRectangle (573,162 84x32), colour toggle: GVL_IO.E_LT_Band_1, colour variable: 16#00555555
        p2167032090: 16#ffc3863c
        p3450524324: 16#00555555
        p3092690914: 16#00555555
    RoundedRectangle (393,164 84x32), colour toggle: GVL_IO.E_LT_Band_2, colour variable: 16#00555555
        p2167032090: 16#ffc3863c
        p3450524324: 16#00555555
        p3092690914: 16#00555555
    RoundedRectangle (202,163 84x32), colour toggle: GVL_IO.E_LT_Band_3, colour variable: 16#00555555
        p2167032090: 16#ffc3863c
        p3450524324: 16#00555555
        p3092690914: 16#00555555
    RoundedRectangle (436,76 24x51)
    RoundedRectangle (420,2 55x78)
    Image (431,105 32x32), invisible if: GVL_HMI.Status_Bohrer_inv, image: VisuSymbols.Symbols.ArrowHalfRightDown
    Image (431,25 32x32), colour toggle: GVL_IO.A_Bohrwerk_zurueck, invisible if: GVL_HMI.Status_BW_Zur_inv, image: VisuSymbols.Symbols.ArrowBoldUp
        p573394764: 16#FF00FF00
        p2175578022: 16#FF000000
    Image (431,30 32x32), invisible if: GVL_HMI.Status_BW_Vor_inv, image: VisuSymbols.Symbols.ArrowBoldDown
    Group (209,71 84x58)
        Label (0,0 84x30), "Werkstücke"
        Rectangle (3,28 36x30), "%d", text variable: PRG_MAIN.fb_Antriebe.FB_Automatik_inst.CTU_Werkstueckzaehler.CV
        Rectangle (47,28 34x30), "%d", text variable: PRG_MAIN.fb_Antriebe.FB_Automatik_inst.CTU_Werkstueckzaehler.PV
        Line (38,49) (50,36)
    Histogram (837,99 735x465), scale format: %.1f, scale 0..100
        p518627256: mm
        p1518820177: GVL_GlobalData.DataArray
        p102497268: GVL_GlobalData.DataArray
        p788070771: ARRAY [0..100] OF DINT
    Button (4,311 150x30)
    Button (14,360 150x30)
    Frame (273,245 377x247)
        shows Page_2()
END_VISUALIZATION
